Yaskawa INFORM job: TEST_13.JBI

/JOB
//NAME TEST_13
///FOLDERNAME INNE
//POS
///NPOS 0,0,0,0,0,0
//INST
///DATE 2023/10/04 15:16
///ATTR SC,RW,RJ
////FRAME ROBOT
///GROUP1 RB1,BS1
///LVARS 0,3,5,0,0,5,0,0
NOP
GETS PX[B000] $PX000
SET LI000 3
SET LI001 1
SUB LI000 LI001
SET I000 LI000
END
